# EPICS substitutions: PIMOT/PIMOT-IOC-01App/Db/asyn_motor.substitutions
file $(MOTOR)/motorApp/Db/asyn_motor.db {

pattern {P,      N,     M,         DTYP,      PORT,  ADDR,    DESC,        EGU,     DIR,  VELO,  VBAS,  ACCL,  BDST,  BVEL,  BACC,  MRES,  PREC,  DHLM,  DLLM,  INIT}
{"\$(P)", 1, "\$(M)", "asynMotor",  "\$(PORT)",    "\$(ADDR)", "HEXAPOD",  mm,  Pos,  10,     0,    .2,    0,     .5,     .2,    0.0001,  6,     125,   -125,  ""}
}
